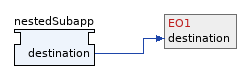
      [picture p97: application DataConnectionTestApp.Test5Solution]
      SUBAPPLICATION nestedSubapp
        VAR_OUTPUT
          destination : BOOL;
        END_VAR
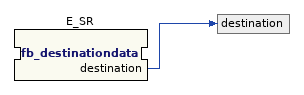
        FBS
          E_SR : fb_destinationdata;
        END_FBS
        DATA_CONNECTIONS
          E_SR.destination TO destination;
        END_CONNECTIONS
      END_SUBAPPLICATION
      DATA_CONNECTIONS
        nestedSubapp.destination TO destination;
      END_CONNECTIONS
    END_SUBAPPLICATION
    SUBAPPLICATION Test6Solution (* crossing connection from FB to nested subapp interface *)
      EVENT_OUTPUT
        EO1;
      END_EVENT
      VAR_OUTPUT
        destination : BOOL;
      END_VAR
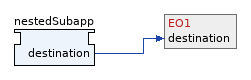
      SUBAPPLICATION nestedSubapp
        VAR_OUTPUT
          destination : BOOL;
        END_VAR
      END_SUBAPPLICATION
      DATA_CONNECTIONS
        nestedSubapp.destination TO destination;
      END_CONNECTIONS
    END_SUBAPPLICATION
    SUBAPPLICATION Test18 (* crossing connection from FB to FB in nested subapp, data pin of same name   &#10;already exists *)
      VAR_OUTPUT
        destination : BOOL;
      END_VAR
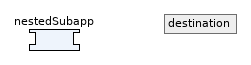
      SUBAPPLICATION nestedSubapp
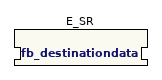
        FBS
          E_SR : fb_destinationdata;
        END_FBS
      END_SUBAPPLICATION
    END_SUBAPPLICATION
    SUBAPPLICATION Test7Solution (* crossing connection from FB to FB in nested subapp, one pin already exists *)
      VAR_OUTPUT
        destination : BOOL;
      END_VAR
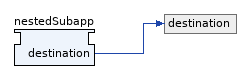
      SUBAPPLICATION nestedSubapp
        VAR_OUTPUT
          destination : BOOL;
        END_VAR
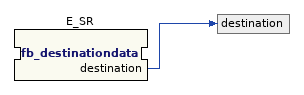
        FBS
          E_SR : fb_destinationdata;
        END_FBS
        DATA_CONNECTIONS
          E_SR.destination TO destination;
        END_CONNECTIONS
      END_SUBAPPLICATION
      DATA_CONNECTIONS
        nestedSubapp.destination TO destination;
      END_CONNECTIONS
    END_SUBAPPLICATION
    SUBAPPLICATION Test8Solution (* crossing connection from FB in subapp to FB in nested subapp *)
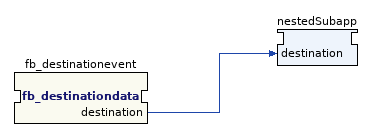
      FBS
        fb_destinationevent : fb_destinationdata;
      END_FBS
      SUBAPPLICATION nestedSubapp
        VAR_INPUT
          destination : BOOL;
        END_VAR
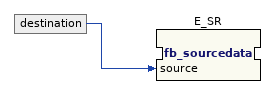
        FBS
          E_SR : fb_sourcedata;
        END_FBS
        DATA_CONNECTIONS
          destination TO E_SR.source;
        END_CONNECTIONS
      END_SUBAPPLICATION
      DATA_CONNECTIONS
        fb_destinationevent.destination TO nestedSubapp.destination;
      END_CONNECTIONS
    END_SUBAPPLICATION
    SUBAPPLICATION SubApp_9
      EVENT_INPUT
        destination;
      END_EVENT
      VAR_INPUT
        destination_1 : BOOL;
      END_VAR
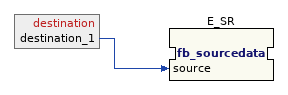
      FBS
        E_SR : fb_sourcedata;
      END_FBS
      DATA_CONNECTIONS
        destination_1 TO E_SR.source;
      END_CONNECTIONS
    END_SUBAPPLICATION
    SUBAPPLICATION Test9Solution (* event input pin already exists outwards *)
      VAR_OUTPUT
        destination : BOOL;
      END_VAR
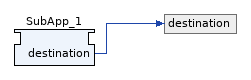
      SUBAPPLICATION SubApp_1
        VAR_OUTPUT
          destination : BOOL;
        END_VAR
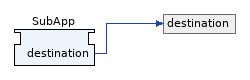
        SUBAPPLICATION SubApp
          VAR_OUTPUT
            destination : BOOL;
          END_VAR
        END_SUBAPPLICATION
        DATA_CONNECTIONS
          SubApp.destination TO destination;
        END_CONNECTIONS
      END_SUBAPPLICATION
      DATA_CONNECTIONS
        SubApp_1.destination TO destination;
      END_CONNECTIONS
    END_SUBAPPLICATION
    SUBAPPLICATION Test10Solution (* data input pin with same name already exists *)
      VAR_OUTPUT
        destination : BOOL;
      END_VAR
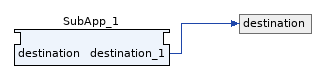
      SUBAPPLICATION SubApp_1
        VAR_INPUT
          destination : INT;
        END_VAR
        VAR_OUTPUT
          destination_1 : BOOL;
        END_VAR
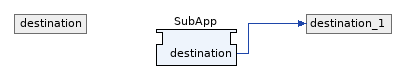
        SUBAPPLICATION SubApp
          VAR_OUTPUT
            destination : BOOL;
          END_VAR
        END_SUBAPPLICATION
        DATA_CONNECTIONS
          SubApp.destination TO destination_1;
        END_CONNECTIONS
      END_SUBAPPLICATION
      DATA_CONNECTIONS
        SubApp_1.destination_1 TO destination;
      END_CONNECTIONS
    END_SUBAPPLICATION
    SUBAPPLICATION SubApp_11
      VAR_INPUT
        source : BOOL;
      END_VAR
    END_SUBAPPLICATION
    SUBAPPLICATION Test11 (* event input pin with same name and incompatible data type already exists *)
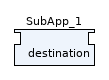
      SUBAPPLICATION SubApp_1
        VAR_OUTPUT
          destination : INT;
        END_VAR
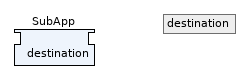
        SUBAPPLICATION SubApp
          VAR_OUTPUT
            destination : BOOL;
          END_VAR
        END_SUBAPPLICATION
      END_SUBAPPLICATION
    END_SUBAPPLICATION
    SUBAPPLICATION SubApp_16
      VAR_INPUT
        source : BOOL;
      END_VAR
    END_SUBAPPLICATION
    SUBAPPLICATION Test11Solution (* event input pin with same name and incompatible data type already exists *)
      VAR_OUTPUT
        destination : BOOL;
      END_VAR
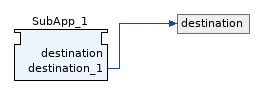
      SUBAPPLICATION SubApp_1
        VAR_OUTPUT
          destination : INT;
          destination_1 : BOOL;
        END_VAR
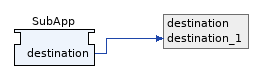
        SUBAPPLICATION SubApp
          VAR_OUTPUT
            destination : BOOL;
          END_VAR
        END_SUBAPPLICATION
        DATA_CONNECTIONS
          SubApp.destination TO destination_1;
        END_CONNECTIONS
      END_SUBAPPLICATION
      DATA_CONNECTIONS
        SubApp_1.destination_1 TO destination;
      END_CONNECTIONS
    END_SUBAPPLICATION
    SUBAPPLICATION SubApp_17
      VAR_INPUT
        source : BOOL;
      END_VAR
    END_SUBAPPLICATION
    SUBAPPLICATION Test12Solution (* event input already exists inwards *)
      VAR_INPUT
        source : INT;
      END_VAR
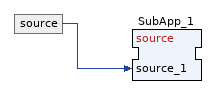
      SUBAPPLICATION SubApp_1
        EVENT_INPUT
          source;
        END_EVENT
        VAR_INPUT
          source_1 : INT;
        END_VAR
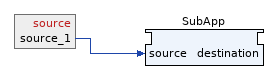
        SUBAPPLICATION SubApp
          VAR_INPUT
            source : INT;
          END_VAR
          VAR_OUTPUT
            destination : INT;
          END_VAR
          DATA_CONNECTIONS
            source TO destination;
          END_CONNECTIONS
        END_SUBAPPLICATION
        DATA_CONNECTIONS
          source_1 TO SubApp.source;
        END_CONNECTIONS
      END_SUBAPPLICATION
      DATA_CONNECTIONS
        source TO SubApp_1.source_1;
      END_CONNECTIONS
    END_SUBAPPLICATION
    SUBAPPLICATION SubApp_13
      VAR_OUTPUT
        source : INT;
      END_VAR
    END_SUBAPPLICATION
    SUBAPPLICATION Test13 (* incompatible data input already exists inwards, skip it *)
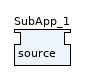
      SUBAPPLICATION SubApp_1
        VAR_INPUT
          source : UINT;
        END_VAR
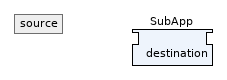
        SUBAPPLICATION SubApp
          VAR_OUTPUT
            destination : INT;
          END_VAR
        END_SUBAPPLICATION
      END_SUBAPPLICATION
    END_SUBAPPLICATION
    SUBAPPLICATION SubApp_18
      VAR_OUTPUT
        source : INT;
      END_VAR
    END_SUBAPPLICATION
    SUBAPPLICATION Test14 (* compatible data input already exists inwards, use it *)
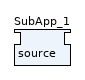
      SUBAPPLICATION SubApp_1
        VAR_INPUT
          source : ANY_INT;
        END_VAR
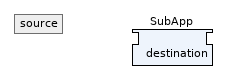
        SUBAPPLICATION SubApp
          VAR_OUTPUT
            destination : UINT;
          END_VAR
        END_SUBAPPLICATION
      END_SUBAPPLICATION
    END_SUBAPPLICATION
    SUBAPPLICATION SubApp_20
      VAR_OUTPUT
        source : UINT;
      END_VAR
    END_SUBAPPLICATION
    SUBAPPLICATION Test15 (* compatible data input already exists inwards, use it *)
      VAR_INPUT
        source : ANY_INT;
      END_VAR
